(* IEC 61131-3 sources: InfiniteStateMachine/extracted_st/infinitestatemachine/functions/issamestate, 1 file *)

(* ---- IsSameState.st ---- *)
(* --- Interface --- *)
FUNCTION IsSameState : BOOL
VAR_INPUT
	itfStateLHS : IState;
	itfStateRHS : IState;
END_VAR
VAR
END_VAR

(* --- Implementation --- *)
IsSameState := itfStateLHS = itfStateRHS;
